TYPE IoStageAxisConfig EXTENDS IoAxisConfig :
STRUCT
END_STRUCT
END_TYPE

(* stored: Version 1.1.0.1, ProductVersion 3.1.4024.12
   DUT IoStageAxisConfig: Id {5cde0062-e600-4e00-b6c4-8571e23f8f4c} *)
